TYPE
Pos2D_t :
STRUCT
    x : DINT;
    y : DINT;
END_STRUCT
END_TYPE

(* stored: Version 1.1.0.1, ProductVersion 3.1.4024.6
   DUT Pos2D_t: Id {412a4c90-bbde-4fda-83df-156dd4f50170} *)
